TYPE ST_EbaraDryPump EXTENDS ST_RoughPump :
STRUCT
(* Extension of the rough pump archetype for ebara 
Applicable to: 
EV-S20
EV-S50
EV-S100
EV-S200
*)

//Controls
q_xMPStart	:	BOOL; //MP (main pump?) start
q_xBPStart	:	BOOL; // Booster pump start (this can be started by the pump automatically)

xBPIlk	:	BOOL;	//Booster pump interlock
rBPIlkSP	:	REAL := 30; //Booster pump pressure setpoint
tonBP	:	TON; //Timer for pressure and valve stability


//Readbacks
i_xMPStatus	:	BOOL; //MP status
i_xBPStatus	:	BOOL; //BP status
i_xWarning	:	BOOL; //Warning status
i_xAlarm	:	BOOL; //Alarm, maps to error
i_xRemote	:	BOOL; //Remote control status


END_STRUCT
END_TYPE

(* stored: Version 1.1.0.1, ProductVersion 3.1.4018.5
   DUT ST_EbaraDryPump: Id {55a0bc2c-4199-48dd-89d3-0255c23678ea} *)
